FUNCTION_BLOCK MIXER (* Mixer Communication Block V1 *)
  (* Standard: 61499-2 *)
  (* Version 1.0, 2023-08-25, ADMIN *)
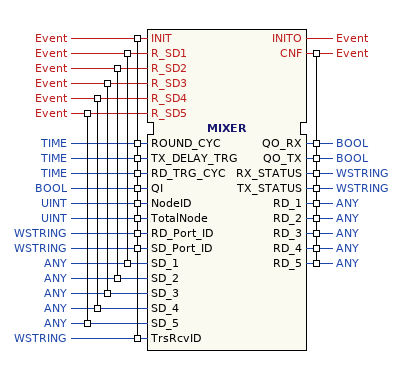
  EVENT_INPUT
    INIT WITH QI, NodeID, TotalNode, TrsRcvID, ROUND_CYC, TX_DELAY_TRG, RD_TRG_CYC, RD_Port_ID, SD_Port_ID; (* Initialization Request *)
    R_SD1 WITH SD_1; (* Normal Execution Request *)
    R_SD2 WITH SD_2;
    R_SD3 WITH SD_3;
    R_SD4 WITH SD_4;
    R_SD5 WITH SD_5;
  END_EVENT
  EVENT_OUTPUT
    INITO; (* Initialization Confirm *)
    CNF WITH QO_RX, RX_STATUS, RD_1, RD_2, RD_3, RD_4, RD_5, TX_STATUS, QO_TX; (* Execution Confirmation *)
  END_EVENT
  VAR_INPUT
    ROUND_CYC : TIME;
    TX_DELAY_TRG : TIME;
    RD_TRG_CYC : TIME;
    QI : BOOL;
    NodeID : UINT;
    TotalNode : UINT;
    RD_Port_ID : WSTRING;
    SD_Port_ID : WSTRING;
    SD_1 : ANY;
    SD_2 : ANY;
    SD_3 : ANY;
    SD_4 : ANY;
    SD_5 : ANY;
    TrsRcvID : WSTRING;
  END_VAR
  VAR_OUTPUT
    QO_RX : BOOL;
    QO_TX : BOOL;
    RX_STATUS : WSTRING;
    TX_STATUS : WSTRING;
    RD_1 : ANY;
    RD_2 : ANY;
    RD_3 : ANY;
    RD_4 : ANY;
    RD_5 : ANY;
  END_VAR
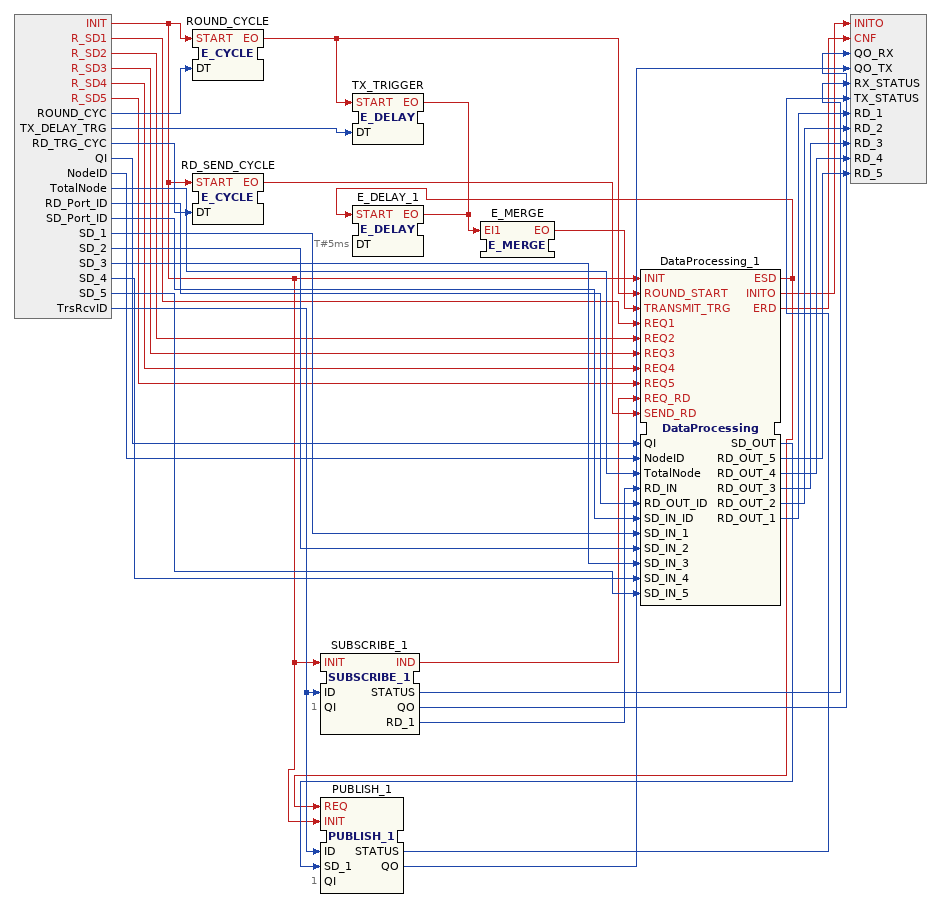
  FBS
    ROUND_CYCLE : E_CYCLE;
    TX_TRIGGER : E_DELAY;
    PUBLISH_1 : PUBLISH_1(QI := 1);
    SUBSCRIBE_1 : SUBSCRIBE_1(QI := 1);
    E_MERGE : E_MERGE;
    DataProcessing_1 : DataProcessing;
    E_DELAY_1 : E_DELAY(DT := T#5ms);
    RD_SEND_CYCLE : E_CYCLE;
  END_FBS
  EVENT_CONNECTIONS
    ROUND_CYCLE.EO TO TX_TRIGGER.START;
    INIT TO DataProcessing_1.INIT;
    ROUND_CYCLE.EO TO DataProcessing_1.ROUND_START;
    DataProcessing_1.ESD TO PUBLISH_1.REQ;
    TX_TRIGGER.EO TO E_MERGE.EI1;
    E_MERGE.EO TO DataProcessing_1.TRANSMIT_TRG;
    E_DELAY_1.EO TO E_MERGE.EI1;
    DataProcessing_1.ESD TO E_DELAY_1.START;
    R_SD1 TO DataProcessing_1.REQ1;
    R_SD2 TO DataProcessing_1.REQ2;
    R_SD3 TO DataProcessing_1.REQ3;
    R_SD4 TO DataProcessing_1.REQ4;
    R_SD5 TO DataProcessing_1.REQ5;
    SUBSCRIBE_1.IND TO DataProcessing_1.REQ_RD;
    INIT TO ROUND_CYCLE.START;
    INIT TO RD_SEND_CYCLE.START;
    INIT TO SUBSCRIBE_1.INIT;
    INIT TO PUBLISH_1.INIT;
    DataProcessing_1.INITO TO INITO;
    RD_SEND_CYCLE.EO TO DataProcessing_1.SEND_RD;
    DataProcessing_1.ERD TO CNF;
  END_CONNECTIONS
  DATA_CONNECTIONS
    SUBSCRIBE_1.STATUS TO RX_STATUS;
    PUBLISH_1.STATUS TO TX_STATUS;
    SUBSCRIBE_1.QO TO QO_RX;
    PUBLISH_1.QO TO QO_TX;
    TrsRcvID TO SUBSCRIBE_1.ID;
    TrsRcvID TO PUBLISH_1.ID;
    DataProcessing_1.SD_OUT TO PUBLISH_1.SD_1;
    QI TO DataProcessing_1.QI;
    NodeID TO DataProcessing_1.NodeID;
    TotalNode TO DataProcessing_1.TotalNode;
    SUBSCRIBE_1.RD_1 TO DataProcessing_1.RD_IN;
    RD_Port_ID TO DataProcessing_1.RD_OUT_ID;
    SD_Port_ID TO DataProcessing_1.SD_IN_ID;
    SD_1 TO DataProcessing_1.SD_IN_1;
    SD_2 TO DataProcessing_1.SD_IN_2;
    SD_3 TO DataProcessing_1.SD_IN_3;
    SD_4 TO DataProcessing_1.SD_IN_4;
    SD_5 TO DataProcessing_1.SD_IN_5;
    RD_TRG_CYC TO RD_SEND_CYCLE.DT;
    ROUND_CYC TO ROUND_CYCLE.DT;
    TX_DELAY_TRG TO TX_TRIGGER.DT;
    DataProcessing_1.RD_OUT_5 TO RD_5;
    DataProcessing_1.RD_OUT_4 TO RD_4;
    DataProcessing_1.RD_OUT_3 TO RD_3;
    DataProcessing_1.RD_OUT_2 TO RD_2;
    DataProcessing_1.RD_OUT_1 TO RD_1;
  END_CONNECTIONS
END_FUNCTION_BLOCK
